(* IEC 61131-3 sources: matiec/tests/bad, 3 files *)

(* ---- end-configuration.st ---- *)
PROGRAM program0
  VAR
    LocalVar0 : DINT;
  END_VAR
  LocalVar0 := 42;
END_PROGRAM

CONFIGURATION config
  RESOURCE resource1 ON PLC
    VAR_GLOBAL
      ResVar0 : DINT;
      ResVar1 : BOOL;
    END_VAR
    TASK task0(INTERVAL := T#20ms,PRIORITY := 0);
    PROGRAM instance0 WITH task0 : program0;
  END_RESOURCE
(* END_CONFIGURATION *)

(* ---- invalid-program-declaration.st ---- *)
PROGRAM
  VAR
    a : REAL;
  END_VAR
  a := 19.4;
END_PROGRAM

(* ---- task-with-zero-time.st ---- *)
PROGRAM program0
  VAR
    LocalVar0 : DINT;
    LocalVar1 : TOD;
  END_VAR

  LocalVar0 := 42;
END_PROGRAM

CONFIGURATION config
  VAR_GLOBAL
    ConfVar0 : DINT;
  END_VAR

  RESOURCE resource1 ON PLC
    (* This leads to FPE in upstream matiec. *)
    TASK task0(INTERVAL := T#0h0m0s0ms,PRIORITY := 1);

    (* Uncomment to build without error: *)
    (* TASK task0(INTERVAL := T#0h0m0s1ms,PRIORITY := 1); *)

    PROGRAM instance0 WITH task0 : program0;
  END_RESOURCE
END_CONFIGURATION
